// TwinCAT 3 PLC project DataTests
// ProgramVersion: 3.1.4024.0
// libraries:
//   Data, * (TomasRompotl)
//   Strings, * (TomasRompotl)
//   Tc2_Standard, * (Beckhoff Automation GmbH)
//   Tc2_System, * (Beckhoff Automation GmbH)
//   Tc3_Module, * (Beckhoff Automation GmbH)
//   TcUnit, * (www.tcunit.org)
//   Types, * (TomasRompotl)
// project tree:
//   / PlcTask.TcTTO
//   Tests/Comparison/ CompareAnyTypeTest.TcPOU, ComparisonFunctionsTest.TcPOU
//   Tests/Manipulate/ ManipulateFunctionsTest.TcPOU
//   Tests/ PRG_Test.TcPOU, TestTableRow.TcDUT (not stored)
//   Tests/QuickSort/ QuickSortFunctionsTest.TcPOU
//   Tests/Sort/ SortFunctionsTest.TcPOU
//   Tests/TableSerialization/ TableDeserializerTest.TcPOU, TableSerializerTest.TcPOU
//   Tests/_TemplateTest/ _TemplateTest.TcPOU (not stored)
// (motion and I/O tree: see PLC project types)
// real-time tasks:
//   TASK BindingTestTask: cycle T#10ms, priority 20, ADS port 350
//   TASK PlcTask: cycle T#10ms, priority 21, ADS port 351
//   TASK PlcTask1: cycle T#10ms, priority 22, ADS port 352
//   TASK PlcTask2: cycle T#10ms, priority 23, ADS port 353

CONFIGURATION DataTests
    RESOURCE PLC ON TwinCAT3
        TASK PlcTask(INTERVAL := T#1ms, PRIORITY := 22);
        PROGRAM PRG_Test WITH PlcTask : PRG_Test;
    END_RESOURCE
END_CONFIGURATION

// ---- Tests/PRG_Test.TcPOU
PROGRAM PRG_Test
VAR
	comparisonFunctionsTest : ComparisonFunctionsTest;
	compareAnyTypeTest : CompareAnyTypeTest;
	
	manipulateFunctionsTest : ManipulateFunctionsTest;
	quickSortFunctionsTest : QuickSortFunctionsTest;
	SortFunctionsTest : SortFunctionsTest;

	tableSerializerTest : TableSerializerTest;
	tableDeserializerTest : TableDeserializerTest;
END_VAR

TcUnit.RUN();

END_PROGRAM

// ---- Tests/Comparison/ComparisonFunctionsTest.TcPOU
FUNCTION_BLOCK ComparisonFunctionsTest EXTENDS TcUnit.FB_TestSuite
VAR
END_VAR

DataEqualsFunction();

METHOD DataEqualsFunction : BOOL
VAR
	data1 : INT;
	data2 : INT;
END_VAR
TcUnit.TEST('Data equals');

data1 := 42;
data2 := 0;

AssertEquals_BOOL(
	Expected := FALSE,
	Actual := DataEquals(data1, data2),
	Message := 'Data should not be equal');

data2 := data1;

AssertEquals_BOOL(
	Expected := TRUE,
	Actual := DataEquals(data1, data2),
	Message := 'Data should be equal');

TEST_FINISHED();
END_METHOD

END_FUNCTION_BLOCK

// ---- Tests/Comparison/CompareAnyTypeTest.TcPOU
FUNCTION_BLOCK CompareAnyTypeTest EXTENDS TcUnit.FB_TestSuite
VAR
END_VAR

IsEqualAnyTypeFunction();
IsGreaterThanAnyTypeFunction();
IsGreaterThanOrEqualAnyTypeFunction();
IsNotEqualAnyTypeFunction();
IsLessThanAnyTypeFunction();
IsLessThanOrEqualAnyTypeFunction();
CompareAnyTypeFunction();

METHOD CompareAnyTypeFunction
VAR  
	data1 : INT := 11;
	data2 : INT := 20; 
END_VAR
TcUnit.TEST('Compare any type function');
 
// Equal
AssertEquals_BOOL(
    Expected := FALSE,
    Actual := CompareAnyType(ToAnyType(data1), ComparisonOperator.Equal, ToAnyType(data2)),
    Message := 'Expected data1 to be less than data2'
);

// NotEqual
AssertEquals_BOOL(
    Expected := TRUE,
    Actual := CompareAnyType(ToAnyType(data1), ComparisonOperator.NotEqual, ToAnyType(data2)),
    Message := 'Expected the two values to be different'
);

// LessThan
AssertEquals_BOOL(
    Expected := TRUE,
    Actual := CompareAnyType(ToAnyType(data1), ComparisonOperator.LessThan, ToAnyType(data2)),
    Message := 'Expected data1 to be less than data2'
);

// LessThanOrEqual
AssertEquals_BOOL(
    Expected := TRUE,
    Actual := CompareAnyType(ToAnyType(data1), ComparisonOperator.LessThanOrEqual, ToAnyType(data2)),
    Message := 'Expected data1 to be less than or equal to data2'
);

// GreaterThan
AssertEquals_BOOL(
    Expected := FALSE,
    Actual := CompareAnyType(ToAnyType(data1), ComparisonOperator.GreaterThan, ToAnyType(data2)),
    Message := 'Expected data1 to be greater than data2'
);

// GreaterThanOrEqual
AssertEquals_BOOL(
    Expected := FALSE,
    Actual := CompareAnyType(ToAnyType(data1), ComparisonOperator.GreaterThanOrEqual, ToAnyType(data2)),
    Message := 'Expected data1 to be greater than or equal to data2'
);

TEST_FINISHED();
END_METHOD

METHOD IsEqualAnyTypeFunction : BOOL
VAR
	data1 : STRING;
	data2 : STRING;
END_VAR
TcUnit.TEST('Is equal any type');

ClearData(data1);
ClearData(data2);
data1 := '';
data2 := 'some test content';

AssertEquals_BOOL(
	Expected := FALSE,
	Actual := CompareAnyType(ToAnyType(data1), ComparisonOperator.Equal, ToAnyType(data2)),
	Message := 'Data should not be equal');

data1 := data2;

AssertEquals_BOOL(
	Expected := TRUE,
	Actual := CompareAnyType(ToAnyType(data1), ComparisonOperator.Equal, ToAnyType(data2)),
	Message := 'Data should be equal');

TEST_FINISHED();
END_METHOD

METHOD IsGreaterThanAnyTypeFunction : BOOL
VAR
	data1 : INT;
	data2 : INT;
END_VAR
TcUnit.TEST('Is greater then any type');

data1 := 5;
data2 := 5;

AssertEquals_BOOL(
	Expected := FALSE,
	Actual := CompareAnyType(ToAnyType(data1), ComparisonOperator.GreaterThan, ToAnyType(data2)),
	Message := 'data1 should not be greater then data2');

data1 := 10;

AssertEquals_BOOL(
	Expected := TRUE,
	Actual := CompareAnyType(ToAnyType(data1), ComparisonOperator.GreaterThan, ToAnyType(data2)),
	Message := 'data1 should be greater then data2');

TEST_FINISHED();
END_METHOD

METHOD IsGreaterThanOrEqualAnyTypeFunction : BOOL
VAR
	data1 : REAL;
	data2 : REAL;
END_VAR
TcUnit.TEST('Is greater then or equal any type');

data1 := 2.14;
data2 := 3.14;

AssertEquals_BOOL(
	Expected := FALSE,
	Actual := CompareAnyType(ToAnyType(data1), ComparisonOperator.GreaterThanOrEqual, ToAnyType(data2)),
	Message := 'data1 should not be greater or equal then data2');

data1 := 3.14;

AssertEquals_BOOL(
	Expected := TRUE,
	Actual := CompareAnyType(ToAnyType(data1), ComparisonOperator.GreaterThanOrEqual, ToAnyType(data2)),
	Message := 'data1 should be equal to data2');

data1 := 4.14;

AssertEquals_BOOL(
	Expected := TRUE,
	Actual := CompareAnyType(ToAnyType(data1), ComparisonOperator.GreaterThanOrEqual, ToAnyType(data2)),
	Message := 'data1 should be greater then data2');

TEST_FINISHED();
END_METHOD

METHOD IsLessThanAnyTypeFunction : BOOL
VAR
	data1 : INT;
	data2 : INT;
END_VAR
TcUnit.TEST('Is less then any type');

data1 := 5;
data2 := 5;

AssertEquals_BOOL(
	Expected := FALSE,
	Actual := CompareAnyType(ToAnyType(data1), ComparisonOperator.LessThan, ToAnyType(data2)),
	Message := 'data1 should not be less then data2');

data1 := 3;

AssertEquals_BOOL(
	Expected := TRUE,
	Actual := CompareAnyType(ToAnyType(data1), ComparisonOperator.LessThan, ToAnyType(data2)),
	Message := 'data1 should be less then data2');

TEST_FINISHED();
END_METHOD

METHOD IsLessThanOrEqualAnyTypeFunction : BOOL
VAR
	data1 : REAL;
	data2 : REAL;
END_VAR
TcUnit.TEST('Is less then or equal any type');

data1 := 4.14;
data2 := 3.14;

AssertEquals_BOOL(
	Expected := FALSE,
	Actual := CompareAnyType(ToAnyType(data1), ComparisonOperator.LessThanOrEqual, ToAnyType(data2)),
	Message := 'data1 should not be less or equal then data2');

data1 := 3.14;

AssertEquals_BOOL(
	Expected := TRUE,
	Actual := CompareAnyType(ToAnyType(data1), ComparisonOperator.LessThanOrEqual, ToAnyType(data2)),
	Message := 'data1 should be equal to data2');

data1 := 2.14;

AssertEquals_BOOL(
	Expected := TRUE,
	Actual := CompareAnyType(ToAnyType(data1), ComparisonOperator.LessThanOrEqual, ToAnyType(data2)),
	Message := 'data1 should be less then data2');

TEST_FINISHED();
END_METHOD

METHOD IsNotEqualAnyTypeFunction : BOOL
VAR
	data1 : STRING;
	data2 : STRING;
END_VAR
TcUnit.TEST('Is not equal any type');

ClearData(data1);
ClearData(data2);
data1 := 'some test content';
data2 := 'some test content';

AssertEquals_BOOL(
	Expected := FALSE,
	Actual := CompareAnyType(ToAnyType(data1), ComparisonOperator.NotEqual, ToAnyType(data2)),
	Message := 'Data should not be equal');

data1 := '';

AssertEquals_BOOL(
	Expected := TRUE,
	Actual := CompareAnyType(ToAnyType(data1), ComparisonOperator.NotEqual, ToAnyType(data2)),
	Message := 'Data should be equal');

TEST_FINISHED();
END_METHOD

END_FUNCTION_BLOCK

// ---- Tests/Manipulate/ManipulateFunctionsTest.TcPOU
FUNCTION_BLOCK ManipulateFunctionsTest EXTENDS TcUnit.FB_TestSuite
VAR
END_VAR

ClearDataFunction();
ShiftDataLeftFunction();
ShiftDataRightFunction();
SwapFunction();
SwapByPointerFunction();
ClearDataAnyTypeFunction();

METHOD ClearDataAnyTypeFunction
VAR 
	intValue : INT;
	stringValue : STRING;
END_VAR
TcUnit.TEST('Clear data any type function');

intValue := 42; 
ClearDataAnyType(ToAnyType(intValue));

AssertEquals_INT(
	Expected := 0,
	Actual := intValue,
	Message := 'Data memory of int type should be all set to 0');
	
stringValue := '42'; 
ClearDataAnyType(ToAnyType(stringValue));
	
AssertEquals_STRING(
	Expected := '',
	Actual := stringValue,
	Message := 'Data memory of string type should be all set to 0');

TEST_FINISHED();
END_METHOD

METHOD ClearDataFunction : BOOL
VAR
	data : INT;
END_VAR
TcUnit.TEST('Clear data function');

data := 42;
ClearData(data);

AssertEquals_INT(
	Expected := 0,
	Actual := data,
	Message := 'Data memory should be all set to 0');

TEST_FINISHED();
END_METHOD

METHOD ShiftDataLeftFunction : BOOL
VAR
	updatedBuffer : ARRAY[0..LastIndex] OF INT;
	
	expected : ARRAY[0..LastIndex] OF INT;
END_VAR
VAR CONSTANT
	LastIndex : INT := 2;
END_VAR
TcUnit.TEST('Shift data left function');

updatedBuffer[LastIndex] := 1;
ShiftDataLeft(updatedBuffer, SIZEOF(INT));
updatedBuffer[LastIndex] := 2;
ShiftDataLeft(updatedBuffer, SIZEOF(INT));
updatedBuffer[LastIndex] := 3;

expected[0] := 1;
expected[1] := 2;
expected[2] := 3;

AssertArrayEquals_INT(
	Expecteds := expected,
	Actuals := updatedBuffer,
	Message := 'Data should be gradually shifter from end to begin');

TEST_FINISHED();
END_METHOD

METHOD ShiftDataRightFunction : BOOL
VAR
	updatedBuffer : ARRAY[0..LastIndex] OF INT;
	
	expected : ARRAY[0..LastIndex] OF INT;
END_VAR
VAR CONSTANT
	LastIndex : INT := 2;
END_VAR
TcUnit.TEST('Shift data right function');

updatedBuffer[0] := 3;
ShiftDataRight(updatedBuffer, SIZEOF(INT));
updatedBuffer[0] := 2;
ShiftDataRight(updatedBuffer, SIZEOF(INT));
updatedBuffer[0] := 1;

expected[0] := 1;
expected[1] := 2;
expected[2] := 3;

AssertArrayEquals_INT(
	Expecteds := expected,
	Actuals := updatedBuffer,
	Message := 'Data should be gradually shifter from begin to end');

TEST_FINISHED();
END_METHOD

METHOD SwapByPointerFunction : BOOL
VAR
	data1 : INT;
	data2 : INT;
END_VAR
TcUnit.TEST('Swap by pointer function');

data1 := 42;
data2 := 420;

SwapByPointer(ADR(data1), ADR(data2), SIZEOF(data1));

AssertEquals_BOOL(
	Expected := TRUE,
	Actual := data1 = 420 AND data2 = 42,
	Message := 'Data should be swapped');

TEST_FINISHED();
END_METHOD

METHOD SwapFunction : BOOL
VAR
	data1 : INT;
	data2 : INT;
END_VAR
TcUnit.TEST('Swap function');

data1 := 42;
data2 := 420;

Swap(data1, data2);

AssertEquals_BOOL(
	Expected := TRUE,
	Actual := data1 = 420 AND data2 = 42,
	Message := 'Data should be swapped');

TEST_FINISHED();
END_METHOD

END_FUNCTION_BLOCK

// ---- Tests/QuickSort/QuickSortFunctionsTest.TcPOU
FUNCTION_BLOCK QuickSortFunctionsTest EXTENDS TcUnit.FB_TestSuite
VAR
END_VAR

QuickSortREALFunction();

METHOD QuickSortREALFunction : BOOL
VAR
	data : ARRAY[0..4] OF REAL;
	expected : ARRAY[0..4] OF REAL;
END_VAR
TcUnit.TEST('QuickSort REAL');

data[0] := 3;
data[1] := 1;
data[2] := 2;
data[3] := 5;
data[4] := 4;

QuickSortREAL(data, 0, 4);

expected[0] := 1;
expected[1] := 2;
expected[2] := 3;
expected[3] := 4;
expected[4] := 5;

AssertArrayEquals_REAL(
	Expecteds := expected,
	Actuals := data,
	Delta := 0.1,
	Message := 'Array should be sorter');

TEST_FINISHED();
END_METHOD

END_FUNCTION_BLOCK

// ---- Tests/Sort/SortFunctionsTest.TcPOU
FUNCTION_BLOCK SortFunctionsTest EXTENDS TcUnit.FB_TestSuite
VAR
END_VAR

SortAnythingFunction();

METHOD SortAnythingFunction : BOOL
VAR
	data : ARRAY[0..4] OF TestTableRow;
	expected : ARRAY[0..4] OF TestTableRow;
	
	i : INT;
END_VAR
TcUnit.TEST('Sort anything');

ClearData(data);
ClearData(expected);

data[0].timestamp := T#3S;
data[0].value1 := 2;
data[0].value2 := 5.555;
data[0].description := 'some text';
data[1].timestamp := T#1S;
data[1].value1 := 8;
data[1].value2 := 3.14;
data[1].description := 'hello world';
data[2].timestamp := T#5S;
data[2].value1 := 15;
data[2].value2 := 9.876;
data[2].description := 'test data';
data[3].timestamp := T#2S;
data[3].value1 := 4;
data[3].value2 := 1.234;
data[3].description := 'sample entry';
data[4].timestamp := T#7S;
data[4].value1 := 11;
data[4].value2 := 6.789;
data[4].description := 'final record';

SortAnything(
	arr := data,
	firstElement := data[0],
	sortBy := data[0].value1,
	order := SortOrder.Descending
);

expected[0].timestamp := T#5S;
expected[0].value1 := 15;
expected[0].value2 := 9.876;
expected[0].description := 'test data';
expected[1].timestamp := T#7S;
expected[1].value1 := 11;
expected[1].value2 := 6.789;
expected[1].description := 'final record';
expected[2].timestamp := T#1S;
expected[2].value1 := 8;
expected[2].value2 := 3.14;
expected[2].description := 'hello world';
expected[3].timestamp := T#2S;
expected[3].value1 := 4;
expected[3].value2 := 1.234;
expected[3].description := 'sample entry';
expected[4].timestamp := T#3S;
expected[4].value1 := 2;
expected[4].value2 := 5.555;
expected[4].description := 'some text';

AssertEquals_BOOL(
	Expected := TRUE,
	Actual := DataEquals(data, expected),
	Message := 'Array should be sorted descending by value1 column');

TEST_FINISHED();
END_METHOD

END_FUNCTION_BLOCK

// ---- Tests/TableSerialization/TableSerializerTest.TcPOU
FUNCTION_BLOCK TableSerializerTest EXTENDS TcUnit.FB_TestSuite
VAR
END_VAR

SerializeTable();
SerializePartOfTableAndSwapColumnsAndWithoutHeader();

METHOD SerializePartOfTableAndSwapColumnsAndWithoutHeader : BOOL
VAR
	table : ARRAY[0..9] OF TestTableRow;
	i : INT;
	
	buffer : STRING(1000);
	sb : StringBuilderExtBuffer := (Buffer := ToAnyType(buffer));
	serializer : TableSerializer := (
		StringBuilder := sb
	);
	
	expected : STRING(1000);
END_VAR
TcUnit.TEST('Serialize part of table and swap columns');

// Prepare data
FOR i := 0 TO 9 DO
	table[i].timestamp := TO_TIME(i);
	table[i].value1 := i;
	table[i].value2 := i * 3.14;
	table[i].description := 'some text';
END_FOR

// Setup serialization
serializer.DecimalSeparator := ',';
serializer.Separator := ';';

// Bind data
serializer.DefineRow(table[0]);
serializer.RowCount := 7;
// Column order is different than structure
serializer.DefineNextColumn(table[0].description);
serializer.DefineNextColumn(table[0].timestamp);
serializer.DefineNextColumn(table[0].value2);

// Serialize
serializer.Serialize(includeHeader := FALSE, clearBuffer := TRUE);

expected := 'some text;T#0ms;0,0$Nsome text;T#1ms;3,14$Nsome text;T#2ms;6,28$Nsome text;T#3ms;9,42$Nsome text;T#4ms;12,56$Nsome text;T#5ms;15,700001$Nsome text;T#6ms;18,84';

AssertEquals_BOOL(
	Expected := TRUE,
	Actual := expected = buffer,
	Message := 'Table was not properly serialized');

TEST_FINISHED();
END_METHOD

METHOD SerializeTable : BOOL
VAR
	table : ARRAY[0..9] OF TestTableRow;
	i : INT;
	
	buffer : STRING(1000);
	sb : StringBuilderExtBuffer := (Buffer := ToAnyType(buffer));
	serializer : TableSerializer := (
		StringBuilder := sb
	);
	
	expected : STRING(1000);
END_VAR
TcUnit.TEST('Serialize table');

// Prepare data
FOR i := 0 TO 9 DO
	table[i].timestamp := TO_TIME(i);
	table[i].value1 := i;
	table[i].value2 := i * 3.14;
	table[i].description := 'some text';
END_FOR

// Setup serialization
serializer.DecimalSeparator := ',';
serializer.Separator := ';';

// Bind data
serializer.DefineRow(table[0]);
serializer.RowCount := 10;
serializer.DefineNextColumnWithName(table[0].timestamp, 'Timestamp');
serializer.DefineNextColumnWithName(table[0].value1, 'Value 1');
serializer.DefineNextColumnWithName(table[0].value2, 'Value 2');
serializer.DefineNextColumnWithName(table[0].description, 'Description');

// Serialize
serializer.Serialize(includeHeader := TRUE, clearBuffer := TRUE);

expected := 'Timestamp;Value 1;Value 2;Description$NT#0ms;0;0,0;some text$NT#1ms;1;3,14;some text$NT#2ms;2;6,28;some text$NT#3ms;3;9,42;some text$NT#4ms;4;12,56;some text$NT#5ms;5;15,700001;some text$NT#6ms;6;18,84;some text$NT#7ms;7;21,98;some text$NT#8ms;8;25,12;some text$NT#9ms;9;28,26;some text';

AssertEquals_BOOL(
	Expected := TRUE,
	Actual := expected = buffer,
	Message := 'Table was not properly serialized');

TEST_FINISHED();
END_METHOD

END_FUNCTION_BLOCK

// ---- Tests/TableSerialization/TableDeserializerTest.TcPOU
FUNCTION_BLOCK TableDeserializerTest EXTENDS TcUnit.FB_TestSuite
VAR
END_VAR

DeserializeTable();
DeserializePartOfTableWithSwappedColumnsAndNoHeader();

METHOD DeserializePartOfTableWithSwappedColumnsAndNoHeader : BOOL
VAR
	data : STRING(1000);
	i : INT;

	table : ARRAY[0..9] OF TestTableRow;
	deserializer : TableDeserializer := (
		DataString := ADR(data)
	);
	
	expected : ARRAY[0..9] OF TestTableRow;
	
	actual : BOOL;
END_VAR
TcUnit.TEST('Deserialize part of table with swapped columns and no header');

// Clear buffers to be able to compare data using memory compare
ClearData(table);
ClearData(expected);

data := 'some text;T#0ms;0,0$Nsome text;T#1ms;3,14$Nsome text;T#2ms;6,28$Nsome text;T#3ms;9,42$Nsome text;T#4ms;12,56$Nsome text;T#5ms;15,700001$Nsome text;T#6ms;18,84$N';

// Define format of data
deserializer.DecimalSeparator := ',';
deserializer.Separator := ';';

// Bind output table
deserializer.DefineRow(table[0]);
deserializer.RowCount := 9;
deserializer.DefineNextColumn(table[0].description);
deserializer.DefineNextColumn(table[0].timestamp);
deserializer.DefineNextColumn(table[0].value2);

// Deserialize
deserializer.Deserialize(includingHeader := FALSE);

// Expected data
FOR i := 0 TO 6 DO
	expected[i].timestamp := TO_TIME(i);
	expected[i].value2 := i * 3.14;
	expected[i].description := 'some text';
END_FOR

actual := TRUE;
FOR i := 0 TO 9 DO
	IF (table[i].timestamp <> expected[i].timestamp
		OR table[i].value1 <> expected[i].value1
		OR ABS(table[i].value2 - expected[i].value2) > 0.1
		OR table[i].description <> expected[i].description) THEN
		
		actual := FALSE;
		EXIT;
	END_IF
END_FOR

AssertEquals_BOOL(
	Expected := TRUE,
	Actual := actual,
	Message := 'Data were not properly deserialized');

TEST_FINISHED();
END_METHOD

METHOD DeserializeTable : BOOL
VAR
	data : STRING(1000);
	i : INT;

	columnNames : ARRAY[0..3] OF T_MaxString;
	table : ARRAY[0..9] OF TestTableRow;
	deserializer : TableDeserializer := (
		DataString := ADR(data)
	);
	
	expected : ARRAY[0..9] OF TestTableRow;
	expectedHeader : ARRAY[0..3] OF T_MaxString;
	
	actual : BOOL;
END_VAR
TcUnit.TEST('Deserialize table');

// Clear buffers to be able to compare data using memory compare
ClearData(columnNames);
ClearData(table);
ClearData(expectedHeader);
ClearData(expected);

data := 'Timestamp;Value 1;Value 2;Description$NT#0ms;0;0,0;some text$NT#1ms;1;3,14;some text$NT#2ms;2;6,28;some text$NT#3ms;3;9,42;some text$NT#4ms;4;12,56;some text$NT#5ms;5;15,700001;some text$NT#6ms;6;18,84;some text$NT#7ms;7;21,98;some text$NT#8ms;8;25,12;some text$NT#9ms;9;28,26;some text';

// Define format of data
deserializer.DecimalSeparator := ',';
deserializer.Separator := ';';

// Bind output table
deserializer.DefineRow(table[0]);
deserializer.RowCount := 10;
deserializer.DefineNextColumn(table[0].timestamp);
deserializer.DefineNextColumn(table[0].value1);
deserializer.DefineNextColumn(table[0].value2);
deserializer.DefineNextColumn(table[0].description);
deserializer.DefineColumnNamesOutput(columnNames);

// Deserialize
deserializer.Deserialize(includingHeader := TRUE);

// Expected data
expectedHeader[0] := 'Timestamp';
expectedHeader[1] := 'Value 1';
expectedHeader[2] := 'Value 2';
expectedHeader[3] := 'Description';
FOR i := 0 TO 9 DO
	expected[i].timestamp := TO_TIME(i);
	expected[i].value1 := i;
	expected[i].value2 := i * 3.14;
	expected[i].description := 'some text';
END_FOR

actual := TRUE;
FOR i := 0 TO 9 DO
	IF (table[i].timestamp <> expected[i].timestamp
		OR table[i].value1 <> expected[i].value1
		OR ABS(table[i].value2 - expected[i].value2) > 0.1
		OR table[i].description <> expected[i].description) THEN
		
		actual := FALSE;
		EXIT;
	END_IF
END_FOR

AssertEquals_BOOL(
	Expected := TRUE,
	Actual := MEMCMP(ADR(columnNames), ADR(expectedHeader), SIZEOF(columnNames)) = 0,
	Message := 'Header was not properly deserialized');
	
AssertEquals_BOOL(
	Expected := TRUE,
	Actual := actual,
	Message := 'Data were not properly deserialized');

TEST_FINISHED();
END_METHOD

END_FUNCTION_BLOCK
